// TIA Portal V21 export
DATA_BLOCK "DiFinal"   // DB102
{ S7_Optimized_Access := 'FALSE' }
// stored: AutoNumber false
   VAR
      ControlKey : Bool;
      EmergencyStop : Bool;
      CompressedAirPressureLow : Bool;
      PowerFailure : Bool;
      PowerReset : Bool;
      MagneticMixerFeedback : Bool;
      CipPumpFeedback : Bool;
      MagneticMixerOverload : Bool;
      CipPumpOverload : Bool;
      RuptureDisc : Bool;
      Cp01FlowSwitch : Bool;
      DiSpare1 : Bool;
      DiSpare2 : Bool;
      MMHighSpeedSensor : Bool;
      DiSpare3 : Bool;
      DiSpare4 : Bool;
      DiSpare5 : Bool;
      DiSpare6 : Bool;
      DiSpare7 : Bool;
      DiSpare8 : Bool;
      DiSpare9 : Bool;
      DiSpare10 : Bool;
   END_VAR
BEGIN
END_DATA_BLOCK
